(* PLC project  *)

PROGRAM P
  VAR
    tmr : TON;
  END_VAR

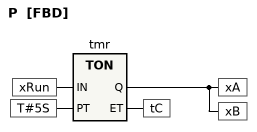
(* FBD diagram, written out as Structured Text *)
tmr(IN := xRun, PT := T#5S);
xA := tmr.Q;
xB := tmr.Q;
tC := tmr.ET;
END_PROGRAM
